(* IEC 61131-3 sources: AdvIecChk/, 3 files *)

(* ---- AdvIecChk.fun ---- *)
(************************************************************************************

Advanced IEC Check Functions Library

File: AdvIecChk.fun
Description: Declaration of library functions

!! Note: See the Automation Studio Help file before modifying these declarations!   !!
!! Most of these functions must be declared exactly as-is in order for the          !!
!! processor to recognize them as check functions. The implementation can change    !!
!! but the declaration cannot!                                                      !!

Authors:
    - Matt Adams (B&R Industrial Automation)
    - Varad Darji (B&R Industrial Automation)
    - Marcus Mangel (B&R Industrial Automation)

************************************************************************************)

FUNCTION CheckDivSint : SINT (*Called before the division/module using a SINT value. Returns the divisor if no errors are found*)
	VAR_INPUT
		divisor : SINT; (*For division: Value that should be divided by. For modulo: Right operand*)
	END_VAR
END_FUNCTION

FUNCTION CheckDivUsint : USINT (*Called before the division/module using a USINT value. Returns the divisor if no errors are found*)
	VAR_INPUT
		divisor : USINT; (*For division: Value that should be divided by. For modulo: Right operand*)
	END_VAR
END_FUNCTION

FUNCTION CheckDivInt : INT (*Called before the division/module using a INT value. Returns the divisor if no errors are found*)
	VAR_INPUT
		divisor : INT; (*For division: Value that should be divided by. For modulo: Right operand*)
	END_VAR
END_FUNCTION

FUNCTION CheckDivUint : UINT (*Called before the division/module using a UINT value. Returns the divisor if no errors are found*)
	VAR_INPUT
		divisor : UINT; (*For division: Value that should be divided by. For modulo: Right operand*)
	END_VAR
END_FUNCTION

FUNCTION CheckDivDint : DINT (*Called before the division/module using a DINT value. Returns the divisor if no errors are found*)
	VAR_INPUT
		divisor : DINT; (*For division: Value that should be divided by. For modulo: Right operand*)
	END_VAR
END_FUNCTION

FUNCTION CheckDivUdint : UDINT (*Called before the division/module using a UDINT value. Returns the divisor if no errors are found*)
	VAR_INPUT
		divisor : UDINT; (*For division: Value that should be divided by. For modulo: Right operand*)
	END_VAR
END_FUNCTION

FUNCTION CheckDivReal : REAL (*Called before the division/module using a REAL value. Returns the divisor if no errors are found*)
	VAR_INPUT
		divisor : REAL; (*For division: Value that should be divided by. For modulo: Right operand*)
	END_VAR
END_FUNCTION

FUNCTION CheckDivLReal : LREAL (*Called before the division/module using a LREAL value. Returns the divisor if no errors are found. (Cannot be used on SG3 or SGC targets)*)
	VAR_INPUT
		divisor : LREAL; (*For division: Value that should be divided by. For modulo: Right operand*)
	END_VAR
END_FUNCTION

FUNCTION CheckBounds : DINT (*Called before accessing an array. Returns the index if no errors are found. Otherwise, returns the problematic index bound*)
	VAR_INPUT
		index : DINT; (*Index being accessed*)
		lower : DINT; (*Lower bound (lowest possible index) of the array*)
		upper : DINT; (*Upper bound (highest possible index) of the array*)
	END_VAR
	VAR
		LowString : STRING[ADVIECCHK_MAX_STRING_LEN]; (*[INTERNAL] Lower bound as a string*)
		UpString : STRING[ADVIECCHK_MAX_STRING_LEN]; (*[INTERNAL] Upper bound as a string*)
		IndexString : STRING[ADVIECCHK_MAX_STRING_LEN]; (*[INTERNAL] Index as a string*)
		ErrorText : STRING[ADVIECCHK_MAX_STRING_LEN]; (*[INTERNAL] Error text created for a long entry based on input data*)
	END_VAR
END_FUNCTION

FUNCTION CheckRange : DINT (*Called before write accessing an enumeration variable. Returns the value if no errors are found. Otherwise, returns the problematic value bound*)
	VAR_INPUT
		value : DINT; (*Enumeration value being accessed*)
		lower : DINT; (*Lower bound (lowest possible value) of the enumeration*)
		upper : DINT; (*Upper bound (highest possible value) of the enumeration*)
	END_VAR
	VAR
		LowString : STRING[ADVIECCHK_MAX_STRING_LEN]; (*[INTERNAL] Lower bound as a string*)
		UpString : STRING[ADVIECCHK_MAX_STRING_LEN]; (*[INTERNAL] Upper bound as a string*)
		ValueString : STRING[ADVIECCHK_MAX_STRING_LEN]; (*[INTERNAL] Value as a string*)
		ErrorText : STRING[ADVIECCHK_MAX_STRING_LEN]; (*[INTERNAL] Error text created for a long entry based on input data*)
	END_VAR
END_FUNCTION

FUNCTION CheckSignedSubrange : DINT (*Called before write access to a variable with the data type "Subrange" if the subrange is used on a signed data type. Returns the value if no errors are found.
Otherwise, returns the problematic value bound*)
	VAR_INPUT
		value : DINT; (*Index being accessed*)
		lower : DINT; (*Lower bound (lowest possible index) of the subrange*)
		upper : DINT; (*Upper bound (highest possible index) of the subrange*)
	END_VAR
	VAR
		LowString : STRING[ADVIECCHK_MAX_STRING_LEN]; (*[INTERNAL] Lower bound as a string*)
		UpString : STRING[ADVIECCHK_MAX_STRING_LEN]; (*[INTERNAL] Lower bound as a string*)
		ValueString : STRING[ADVIECCHK_MAX_STRING_LEN]; (*[INTERNAL] Value as a string*)
		ErrorText : STRING[ADVIECCHK_MAX_STRING_LEN]; (*[INTERNAL] Error text created for a long entry based on input data*)
	END_VAR
END_FUNCTION

FUNCTION CheckUnsignedSubrange : UDINT (*Called before write access to a variable with the data type "Subrange" if the subrange is used on an unsigned data type. Returns the value if no errors are found.
Otherwise, returns the problematic value bound*)
	VAR_INPUT
		value : UDINT; (*Index being accessed*)
		lower : UDINT; (*Lower bound (lowest possible index) of the subrange*)
		upper : UDINT; (*Upper bound (highest possible index) of the subrange*)
	END_VAR
	VAR
		LowString : STRING[ADVIECCHK_MAX_STRING_LEN]; (*[INTERNAL] Lower bound as a string*)
		UpString : STRING[ADVIECCHK_MAX_STRING_LEN]; (*[INTERNAL] Upper bound as a string*)
		ValueString : STRING[ADVIECCHK_MAX_STRING_LEN]; (*[INTERNAL] Value as a string*)
		ErrorText : STRING[ADVIECCHK_MAX_STRING_LEN]; (*[INTERNAL] Error text created for a long entry based on input data*)
	END_VAR
END_FUNCTION

FUNCTION CheckReadAccess : UDINT (*Called before (read) accessing a memory address using a dynamic variable (ADR). Returns the input address*)
	VAR_INPUT
		address : UDINT; (*Address of the memory area being accessed*)
	END_VAR
END_FUNCTION

FUNCTION CheckWriteAccess : UDINT (*Called before (write) accessing a memory address using a dynamic variable (ADR). Returns the input address*)
	VAR_INPUT
		address : UDINT; (*Address of the memory area being accessed*)
	END_VAR
END_FUNCTION

FUNCTION MakeEntry : UDINT (*Creates a Logger entry detailing any errors. Returns a pointer to out_text*)
	VAR_INPUT
		ErrorCode : UINT; (*Error code that is used to generate a logbook Entry ID. Valid values are 0 to 65535*)
		ErrorText : STRING[ADVIECCHK_MAX_STRING_LEN]; (*Message string for the logbook. Additional characters will be added by the function before publishing the logbook entry*)
	END_VAR
	VAR
		taskname : STRING[ADVIECCHK_MAX_STRING_LEN]; (*[INTERNAL] Name of the task which caused the error. From ST_name()*)
		group : USINT; (*[INTERNAL] Task group number - See docs for ST_name in sys_lib. This will always be zero*)
		status_name : UINT; (*[INTERNAL] Return status of ST_name()*)
		out_text : STRING[ADVIECCHK_MAX_STRING_LEN]; (*[INTERNAL] Final error message text that is written to the logbook. Must be null terminated and maximum 32 characters (see ERRxwarning() docs)*)
		error_facility : UINT; (*[INTERNAL] Facility used to create the log Event ID. See ArEventLog documentation*)
		fb_ArEventLogGetIdent : ArEventLogGetIdent; (*[INTERNAL] Function block to get the ident of a logbook*)
		fb_ArEventLogWrite : ArEventLogWrite; (*[INTERNAL] Function block to write a log entry to the logbook*)
	END_VAR
END_FUNCTION

FUNCTION StrCatToMaxLen : UDINT (*Concatenates two strings, but keeps the result under the max allowed length. Also ensures the the string ends in a zero (null). Returns the length of the new string*)
	VAR_INPUT
		pDest : UDINT; (*Address of the destination string (will be modified)*)
		pSrc : UDINT; (*Address of the source string (not modified)*)
		MaxLength : UDINT; (*Maximum character length of the destination string*)
	END_VAR
	VAR
		destLen : UDINT; (*[INTERNAL] Holds the length of the string at pDest*)
		srcLen : UDINT; (*[INTERNAL] Holds the length of the string at pSrc*)
		lenToCopy : UDINT; (*[INTERNAL] Number of bytes to be copied, in the case of a partial string*)
	END_VAR
END_FUNCTION

(* ---- AdvIecChk.st ---- *)
(************************************************************************************

Advanced IEC Check Functions Library

File: AdvIecChk.st
Description: Implentation of library functions
Authors:
    - Matt Adams (B&R Industrial Automation)
    - Varad Darji (B&R Industrial Automation)
    - Marcus Mangel (B&R Industrial Automation)

************************************************************************************)

(* Called before the division/module using a SINT value. Returns the divisor if no errors are found *)
(* Replaces CheckDivByte, which may return incorrect results *)
FUNCTION CheckDivSint

    IF divisor=0 THEN
        CheckDivSint := 1;
        MakeEntry(55555,'SINT division by 0');
    ELSE
        CheckDivSint := divisor;
    END_IF

END_FUNCTION

(* Called before the division/module using a USINT value. Returns the divisor if no errors are found *)
(* Replaces CheckDivByte, which may return incorrect results *)
FUNCTION CheckDivUsint

    IF divisor=0 THEN
        CheckDivUsint := 1;
        MakeEntry(55555,'USINT division by 0');
    ELSE
        CheckDivUsint := divisor;
    END_IF

END_FUNCTION

(* Called before the division/module using an INT value. Returns the divisor if no errors are found *)
(* Replaces CheckDivWord, which may return incorrect results *)
FUNCTION CheckDivInt

    IF divisor=0 THEN
        CheckDivInt := 1;
        MakeEntry(55555,'INT division by 0');
    ELSE
        CheckDivInt := divisor;
    END_IF

END_FUNCTION

(* Called before the division/module using a UINT value. Returns the divisor if no errors are found *)
(* Replaces CheckDivWord, which may return incorrect results *)
FUNCTION CheckDivUint

    IF divisor=0 THEN
        CheckDivUint := 1;
        MakeEntry(55555,'UINT division by 0');
    ELSE
        CheckDivUint := divisor;
    END_IF

END_FUNCTION

(* Called before the division/module using a DINT value. Returns the divisor if no errors are found *)
(* Replaces CheckDivDWord, which may return incorrect results *)
FUNCTION CheckDivDint

    IF divisor=0 THEN
        CheckDivDint := 1;
        MakeEntry(55555,'DINT division by 0');
    ELSE
        CheckDivDint := divisor;
    END_IF

END_FUNCTION

(* Called before the division/module using a UDINT value. Returns the divisor if no errors are found *)
(* Replaces CheckDivDWord, which may return incorrect results *)
FUNCTION CheckDivUdint

    IF divisor=0 THEN
        CheckDivUdint := 1;
        MakeEntry(55555,'UDINT division by 0');
    ELSE
        CheckDivUdint := divisor;
    END_IF

END_FUNCTION

(* Called before the division/module using a REAL value. Returns the divisor if no errors are found *)
FUNCTION CheckDivReal

    IF divisor=0 THEN
        CheckDivReal := 1;
        MakeEntry(55555,'REAL division by 0');
    ELSE
        CheckDivReal := divisor;
    END_IF

END_FUNCTION

(* Called before the division/module using a LREAL value. Returns the divisor if no errors are found *)
(* CANNOT BE USED on SG3 OR SGC targets!! *)
FUNCTION CheckDivLReal

    IF divisor=0 THEN
        CheckDivLReal := 1;
        MakeEntry(55555,'LREAL division by 0');
    ELSE
        CheckDivLReal := divisor;
    END_IF

END_FUNCTION

(* Called before accessing an array. Returns the index if no errors are found.
Otherwise, returns the problematic index bound *)
FUNCTION CheckBounds

    IF index < lower THEN
        CheckBounds := lower; // Unless: See end of function
        brsitoa(lower, ADR(LowString));
        brsitoa(upper, ADR(UpString));
        brsitoa(index, ADR(IndexString));
        brsstrcpy(ADR(ErrorText),ADR('Array Index '));
        StrCatToMaxLen(ADR(ErrorText),ADR(IndexString),ADVIECCHK_MAX_STRING_LEN);
        StrCatToMaxLen(ADR(ErrorText),ADR(' is outside range ['),ADVIECCHK_MAX_STRING_LEN);
        StrCatToMaxLen(ADR(ErrorText),ADR(LowString),ADVIECCHK_MAX_STRING_LEN);
        StrCatToMaxLen(ADR(ErrorText),ADR('..'),ADVIECCHK_MAX_STRING_LEN);
        StrCatToMaxLen(ADR(ErrorText),ADR(UpString),ADVIECCHK_MAX_STRING_LEN);
        StrCatToMaxLen(ADR(ErrorText),ADR(']'),ADVIECCHK_MAX_STRING_LEN);
        MakeEntry(55555,ErrorText);
    ELSIF index > upper THEN
        CheckBounds := upper; // Unless: See end of function
        brsitoa(lower, ADR(LowString));
        brsitoa(upper, ADR(UpString));
        brsitoa(index, ADR(IndexString));
        brsstrcpy(ADR(ErrorText),ADR('Array Index '));
        StrCatToMaxLen(ADR(ErrorText),ADR(IndexString),ADVIECCHK_MAX_STRING_LEN);
        StrCatToMaxLen(ADR(ErrorText),ADR(' is outside range ['),ADVIECCHK_MAX_STRING_LEN);
        StrCatToMaxLen(ADR(ErrorText),ADR(LowString),ADVIECCHK_MAX_STRING_LEN);
        StrCatToMaxLen(ADR(ErrorText),ADR('..'),ADVIECCHK_MAX_STRING_LEN);
        StrCatToMaxLen(ADR(ErrorText),ADR(UpString),ADVIECCHK_MAX_STRING_LEN);
        StrCatToMaxLen(ADR(ErrorText),ADR(']'),ADVIECCHK_MAX_STRING_LEN);
        MakeEntry(55555,ErrorText);
    ELSE
        CheckBounds := index;
    END_IF

    #if defined(_CHECKLIB_KEEP_INDEX_VALUES)
    // Don't modify accessed index
    // This may lead to undefined behavior!
    CheckBounds := index;
    #endif

END_FUNCTION

(* Called before write accessing an enumeration variable. Returns the value if no errors are found.
Otherwise, returns the problematic value bound *)
FUNCTION CheckRange

    IF value < lower THEN
        CheckRange := lower; // Unless: See end of function
        brsitoa(lower, ADR(LowString));
        brsitoa(upper, ADR(UpString));
        brsitoa(value, ADR(ValueString));
        brsstrcpy(ADR(ErrorText),ADR('Enumeration Value '));
        StrCatToMaxLen(ADR(ErrorText),ADR(ValueString),ADVIECCHK_MAX_STRING_LEN);
        StrCatToMaxLen(ADR(ErrorText),ADR(' is outside range ['),ADVIECCHK_MAX_STRING_LEN);
        StrCatToMaxLen(ADR(ErrorText),ADR(LowString),ADVIECCHK_MAX_STRING_LEN);
        StrCatToMaxLen(ADR(ErrorText),ADR('..'),ADVIECCHK_MAX_STRING_LEN);
        StrCatToMaxLen(ADR(ErrorText),ADR(UpString),ADVIECCHK_MAX_STRING_LEN);
        StrCatToMaxLen(ADR(ErrorText),ADR(']'),ADVIECCHK_MAX_STRING_LEN);
        MakeEntry(55555,ErrorText);
    ELSIF value > upper THEN
        CheckRange := upper; // Unless: See end of function
        brsitoa(lower, ADR(LowString));
        brsitoa(upper, ADR(UpString));
        brsitoa(value, ADR(ValueString));
        brsstrcpy(ADR(ErrorText),ADR('Enumeration Value '));
        StrCatToMaxLen(ADR(ErrorText),ADR(ValueString),ADVIECCHK_MAX_STRING_LEN);
        StrCatToMaxLen(ADR(ErrorText),ADR(' is outside range ['),ADVIECCHK_MAX_STRING_LEN);
        StrCatToMaxLen(ADR(ErrorText),ADR(LowString),ADVIECCHK_MAX_STRING_LEN);
        StrCatToMaxLen(ADR(ErrorText),ADR('..'),ADVIECCHK_MAX_STRING_LEN);
        StrCatToMaxLen(ADR(ErrorText),ADR(UpString),ADVIECCHK_MAX_STRING_LEN);
        StrCatToMaxLen(ADR(ErrorText),ADR(']'),ADVIECCHK_MAX_STRING_LEN);
        MakeEntry(55555,ErrorText);
    ELSE
        CheckRange := value;
    END_IF

    #if defined(_CHECKLIB_KEEP_INDEX_VALUES)
    // Don't modify accessed value
    // This may lead to undefined behavior!
    CheckRange := value;
    #endif

END_FUNCTION

(* Called before write access to a variable with the data type "Subrange" if the subrange is used on a signed data type. Returns the value if no errors are found.
Otherwise, returns the problematic value bound *)
FUNCTION CheckSignedSubrange

    IF value < lower THEN
        CheckSignedSubrange := lower; // Unless: See end of function
        brsitoa(lower, ADR(LowString));
        brsitoa(upper, ADR(UpString));
        brsitoa(value, ADR(ValueString));
        brsstrcpy(ADR(ErrorText),ADR('Signed Subrange Index '));
        StrCatToMaxLen(ADR(ErrorText),ADR(ValueString),ADVIECCHK_MAX_STRING_LEN);
        StrCatToMaxLen(ADR(ErrorText),ADR(' is outside range ['),ADVIECCHK_MAX_STRING_LEN);
        StrCatToMaxLen(ADR(ErrorText),ADR(LowString),ADVIECCHK_MAX_STRING_LEN);
        StrCatToMaxLen(ADR(ErrorText),ADR('..'),ADVIECCHK_MAX_STRING_LEN);
        StrCatToMaxLen(ADR(ErrorText),ADR(UpString),ADVIECCHK_MAX_STRING_LEN);
        StrCatToMaxLen(ADR(ErrorText),ADR(']'),ADVIECCHK_MAX_STRING_LEN);
        MakeEntry(55555,ErrorText);
    ELSIF value > upper THEN
        CheckSignedSubrange := upper; // Unless: See end of function
        brsitoa(lower, ADR(LowString));
        brsitoa(upper, ADR(UpString));
        brsitoa(value, ADR(ValueString));
        StrCatToMaxLen(ADR(ErrorText),ADR('Signed Subrange Index '),ADVIECCHK_MAX_STRING_LEN);
        StrCatToMaxLen(ADR(ErrorText),ADR(ValueString),ADVIECCHK_MAX_STRING_LEN);
        StrCatToMaxLen(ADR(ErrorText),ADR(' is outside range ['),ADVIECCHK_MAX_STRING_LEN);
        StrCatToMaxLen(ADR(ErrorText),ADR(LowString),ADVIECCHK_MAX_STRING_LEN);
        StrCatToMaxLen(ADR(ErrorText),ADR('..'),ADVIECCHK_MAX_STRING_LEN);
        StrCatToMaxLen(ADR(ErrorText),ADR(UpString),ADVIECCHK_MAX_STRING_LEN);
        StrCatToMaxLen(ADR(ErrorText),ADR(']'),ADVIECCHK_MAX_STRING_LEN);
        MakeEntry(55555,ErrorText);
    ELSE
        CheckSignedSubrange := value;
    END_IF

    #if defined(_CHECKLIB_KEEP_INDEX_VALUES)
    // Don't modify accessed value
    // This may lead to undefined behavior!
    CheckSignedSubrange := value;
    #endif

END_FUNCTION

(* Called before write access to a variable with the data type "Subrange" if the subrange is used on an unsigned data type. Returns the value if no errors are found.
Otherwise, returns the problematic value bound *)
FUNCTION CheckUnsignedSubrange

    IF value < lower THEN
        CheckUnsignedSubrange := lower; // Unless: See end of function
        brsitoa(lower, ADR(LowString));
        brsitoa(upper, ADR(UpString));
        brsitoa(value, ADR(ValueString));
        brsstrcpy(ADR(ErrorText),ADR('Unsigned Subrange Index '));
        StrCatToMaxLen(ADR(ErrorText),ADR(ValueString),ADVIECCHK_MAX_STRING_LEN);
        StrCatToMaxLen(ADR(ErrorText),ADR(' is outside range ['),ADVIECCHK_MAX_STRING_LEN);
        StrCatToMaxLen(ADR(ErrorText),ADR(LowString),ADVIECCHK_MAX_STRING_LEN);
        StrCatToMaxLen(ADR(ErrorText),ADR('..'),ADVIECCHK_MAX_STRING_LEN);
        StrCatToMaxLen(ADR(ErrorText),ADR(UpString),ADVIECCHK_MAX_STRING_LEN);
        StrCatToMaxLen(ADR(ErrorText),ADR(']'),ADVIECCHK_MAX_STRING_LEN);
        MakeEntry(55555,ErrorText);
    ELSIF value > upper THEN
        CheckUnsignedSubrange := upper; // Unless: See end of function
        brsitoa(lower, ADR(LowString));
        brsitoa(upper, ADR(UpString));
        brsitoa(value, ADR(ValueString));
        brsstrcpy(ADR(ErrorText),ADR('Unsigned Subrange Index '));
        StrCatToMaxLen(ADR(ErrorText),ADR(ValueString),ADVIECCHK_MAX_STRING_LEN);
        StrCatToMaxLen(ADR(ErrorText),ADR(' is outside range ['),ADVIECCHK_MAX_STRING_LEN);
        StrCatToMaxLen(ADR(ErrorText),ADR(LowString),ADVIECCHK_MAX_STRING_LEN);
        StrCatToMaxLen(ADR(ErrorText),ADR('..'),ADVIECCHK_MAX_STRING_LEN);
        StrCatToMaxLen(ADR(ErrorText),ADR(UpString),ADVIECCHK_MAX_STRING_LEN);
        StrCatToMaxLen(ADR(ErrorText),ADR(']'),ADVIECCHK_MAX_STRING_LEN);
        MakeEntry(55555,ErrorText);
    ELSE
        CheckUnsignedSubrange := value;
    END_IF

    #if defined(_CHECKLIB_KEEP_INDEX_VALUES)
    // Don't modify accessed value
    // This may lead to undefined behavior!
    CheckUnsignedSubrange := value;
    #endif

END_FUNCTION

(* Called before (read) accessing a memory address using a dynamic variable (ADR). Returns the input address *)
// Note: We cannot substitute in any addresses here
// This always returns a zero address
// That means a pagefault will occur no matter what, but at least we can log why
FUNCTION CheckReadAccess

    IF address=0 THEN
        MakeEntry(55555,'Read from memory address of zero');
        CheckReadAccess:=0;
    ELSE
        CheckReadAccess:=address;
    END_IF

END_FUNCTION

(* Called before (write) accessing a memory address using a dynamic variable (ADR). Returns the input address *)
// Note: We cannot substitute in any addresses here
// This always returns a zero address
// That means a pagefault will occur no matter what, but at least we can log why
FUNCTION CheckWriteAccess

    IF address=0 THEN
        MakeEntry(55555,'Write to memory address of zero');
        CheckWriteAccess:=0;
    ELSE
        CheckWriteAccess:=address;
    END_IF

END_FUNCTION

(* Creates a Logger entry detailing any errors. Returns a pointer to out_text *)
FUNCTION MakeEntry

    // Get task name and add to error text string
    status_name := ST_name(0,ADR(taskname),ADR(group));

    brsmemset(ADR(out_text),0,SIZEOF(out_text)); // We need to make sure the data is null terminated, so start with all zeros
    StrCatToMaxLen(ADR(out_text),ADR(ErrorText), ADVIECCHK_MAX_STRING_LEN);

    IF status_name = 0 THEN
        StrCatToMaxLen(ADR(out_text),ADR(' in task '), ADVIECCHK_MAX_STRING_LEN);
        StrCatToMaxLen(ADR(out_text),ADR('"'), ADVIECCHK_MAX_STRING_LEN);
        StrCatToMaxLen(ADR(out_text),ADR(taskname), ADVIECCHK_MAX_STRING_LEN);
        StrCatToMaxLen(ADR(out_text),ADR('"'), ADVIECCHK_MAX_STRING_LEN);
    END_IF;

    // Finalize logbook entry - Write to the existing User logbook
    // It would be possible to create our own logbook, but that would be much more complex
    error_facility := 0; // See ArEventLog documentation on the 32-bit event ID

    fb_ArEventLogGetIdent.Execute := TRUE;
    fb_ArEventLogGetIdent.Name := '$$arlogusr'; // This is the only system logbook we can access
    fb_ArEventLogGetIdent();

    fb_ArEventLogWrite.Execute := TRUE;
    fb_ArEventLogWrite.Ident := fb_ArEventLogGetIdent.Ident;
    fb_ArEventLogWrite.EventID := ArEventLogMakeEventID(arEVENTLOG_SEVERITY_ERROR,error_facility,ErrorCode);
    fb_ArEventLogWrite.AddData := ADR(out_text);
    fb_ArEventLogWrite.AddDataFormat := arEVENTLOG_ADDFORMAT_TEXT;
    fb_ArEventLogWrite.AddDataSize := MIN(SIZEOF(out_text),brsstrlen(ADR(out_text))+1); // If string doesn't fill the whole buffer, take just it's length
    fb_ArEventLogWrite.ObjectID := 'AdvIecChk';                                         // plus the next char (should be a zero, this is the trailing null char)
    fb_ArEventLogWrite();

    MakeEntry := brsstrlen(ADR(out_text));

    #if defined(_CHECKLIB_FORCE_RESTART)
    brsmemcpy(1,1,1); // Create a pagefault on purpose to get the backtrace data
    #endif

END_FUNCTION

(* Concatenates two strings, but keeps the result under the max allowed length.
Also ensures the the string ends in a zero (null).
Returns the length of the new string *)
FUNCTION StrCatToMaxLen

    IF (pDest = 0) OR (pSrc = 0) OR (MaxLength = 0) THEN
        StrCatToMaxLen := 0;
        RETURN;
    END_IF;

    destLen := brsstrlen(pDest);
    srcLen := brsstrlen(pSrc);

    lenToCopy := MIN(srcLen,(MaxLength - destLen)); // Copy the full src string if possible, otherwise copy a partial string
    brsmemcpy(pDest + destLen, pSrc, lenToCopy);
    brsmemset(pDest + destLen + lenToCopy, 0, 1); // Ensure trailing null character
    StrCatToMaxLen := destLen + lenToCopy;

END_FUNCTION

(* ---- AdvIecChk.var ---- *)
(************************************************************************************

Advanced IEC Check Functions Library

File: AdvIecChk.var
Description: Constants used in the AdvIecChk library
Authors:
    - Marcus Mangel (B&R Industrial Automation)

************************************************************************************)
VAR CONSTANT
	ADVIECCHK_MAX_STRING_LEN : USINT := 64; (*Maximum character length for the error info string. Used to prevent buffer overflow*)
END_VAR
